(* Logix 5000 project; controller DispersionPlc vendor 1 type 14 code 108 rev 34.11; software revision 34.01; part 21 of 22 *)
(* tags used below, declared in another part *)
   DummyOutput : BOOL;
   Estop_Disp : ALIAS FOR Local:3:I.Data.1;
   FIT_4305_xx : AStd_AnalogInput;
   GenPurp : AStd_GeneralPurp;
   LS_4302_High : BOOL;
   SV_4307_1 : AStd_VlvOC;
   SV_4307_1_AOI : AStd_VlvOC_AOI;
   T0110_PhaseTimedAgitate : AStd_PLI;
   TIT_4305_1 : AStd_AnalogInput;
   TIT_4307_1 : AStd_AnalogInput;
   TIT_4307_1_AOI : AStd_AI_AOI;
   V4307_PhaseAddRO : AStd_PLI;
   V4307_PhaseAddRO_AOI : AStd_PLI_AOI;
   V4307_PhaseAgitation : AStd_PLI;
   V4307_PhaseAgitation_AOI : AStd_PLI_AOI;
   VFD_4307_1 : AStd_VFD;
   VFD_4307_1_AOI : AStd_VFD_AOI;
   WIT_4302_1 : AStd_AnalogInput;
   WIT_4307_1 : AStd_AnalogInput;
   WIT_4307_1_AOI : AStd_AI_AOI;
   XV_4301_8 : AStd_VlvOC;
   XV_4302_10 : AStd_VlvOC;
   XV_4302_8 : AStd_VlvOC;
   XV_4306_3 : AStd_VlvOC;
   XV_4306_5 : AStd_VlvOC;
   XV_4307_1 : AStd_VlvOC;
   XV_4307_1_AOI : AStd_VlvOC_AOI;
   XV_4307_1_IOpn : BOOL;
   XV_4307_1_OCls : BOOL;
   XV_4307_2 : AStd_VlvOC;
   XV_4307_2_AOI : AStd_VlvOC_AOI;
   XV_4307_2_IOpn : BOOL;
   XV_4307_2_OCls : BOOL;
   XV_4307_3 : AStd_VlvOC;
   XV_4307_3_AOI : AStd_VlvOC_AOI;
   XV_4307_3_IOpn : BOOL;
   XV_4307_3_OCls : BOOL;
   XV_4307_4 : AStd_VlvOC;
   XV_4307_4_AOI : AStd_VlvOC_AOI;
   XV_4307_4_IOpn : BOOL;
   XV_4307_4_OCls : BOOL;
   XV_4307_6 : AStd_VlvOC;
   XV_4307_6_AOI : AStd_VlvOC_AOI;
   XV_4307_6_IOpn : BOOL;
   XV_4307_6_OCls : BOOL;

PROGRAM Unit_V4307   (* main routine MainRoutine *)

ROUTINE Device_SV_4307_1   (* ladder *)
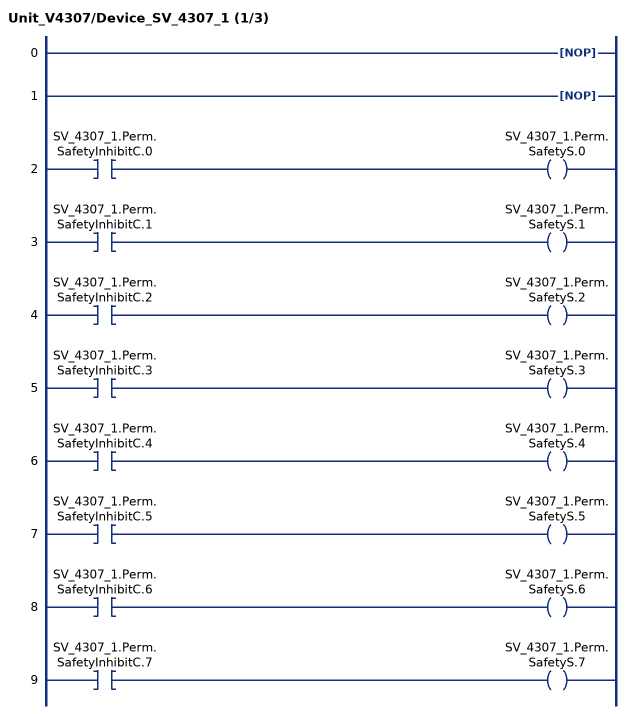
   0: NOP();
   1: NOP();
   2: XIC(SV_4307_1.Perm.SafetyInhibitC.0)OTE(SV_4307_1.Perm.SafetyS.0);
   3: XIC(SV_4307_1.Perm.SafetyInhibitC.1)OTE(SV_4307_1.Perm.SafetyS.1);
   4: XIC(SV_4307_1.Perm.SafetyInhibitC.2)OTE(SV_4307_1.Perm.SafetyS.2);
   5: XIC(SV_4307_1.Perm.SafetyInhibitC.3)OTE(SV_4307_1.Perm.SafetyS.3);
   6: XIC(SV_4307_1.Perm.SafetyInhibitC.4)OTE(SV_4307_1.Perm.SafetyS.4);
   7: XIC(SV_4307_1.Perm.SafetyInhibitC.5)OTE(SV_4307_1.Perm.SafetyS.5);
   8: XIC(SV_4307_1.Perm.SafetyInhibitC.6)OTE(SV_4307_1.Perm.SafetyS.6);
   9: XIC(SV_4307_1.Perm.SafetyInhibitC.7)OTE(SV_4307_1.Perm.SafetyS.7);
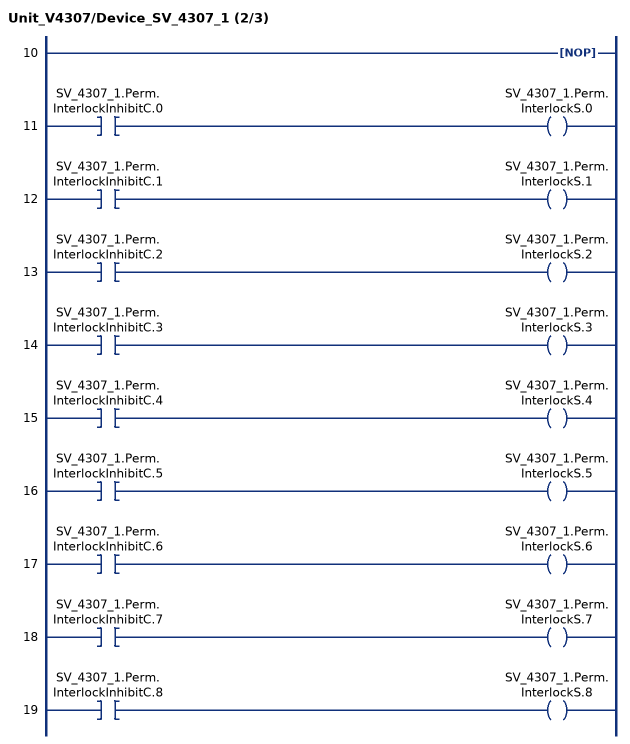
   10: NOP();
   11: XIC(SV_4307_1.Perm.InterlockInhibitC.0)OTE(SV_4307_1.Perm.InterlockS.0);
   12: XIC(SV_4307_1.Perm.InterlockInhibitC.1)OTE(SV_4307_1.Perm.InterlockS.1);
   13: XIC(SV_4307_1.Perm.InterlockInhibitC.2)OTE(SV_4307_1.Perm.InterlockS.2);
   14: XIC(SV_4307_1.Perm.InterlockInhibitC.3)OTE(SV_4307_1.Perm.InterlockS.3);
   15: XIC(SV_4307_1.Perm.InterlockInhibitC.4)OTE(SV_4307_1.Perm.InterlockS.4);
   16: XIC(SV_4307_1.Perm.InterlockInhibitC.5)OTE(SV_4307_1.Perm.InterlockS.5);
   17: XIC(SV_4307_1.Perm.InterlockInhibitC.6)OTE(SV_4307_1.Perm.InterlockS.6);
   18: XIC(SV_4307_1.Perm.InterlockInhibitC.7)OTE(SV_4307_1.Perm.InterlockS.7);
   19: XIC(SV_4307_1.Perm.InterlockInhibitC.8)OTE(SV_4307_1.Perm.InterlockS.8);
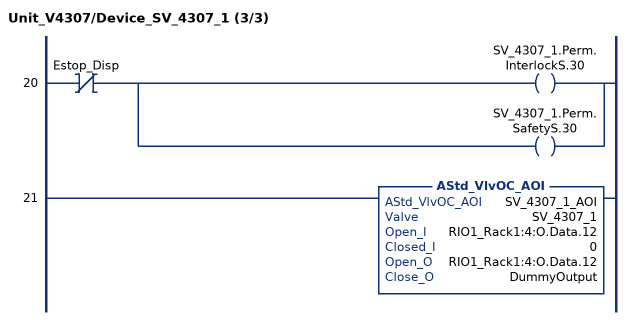
   20: XIO(Estop_Disp)[OTE(SV_4307_1.Perm.InterlockS.30) ,OTE(SV_4307_1.Perm.SafetyS.30) ];
   21: AStd_VlvOC_AOI(SV_4307_1_AOI,SV_4307_1,RIO1_Rack1:4:O.Data.12,0,RIO1_Rack1:4:O.Data.12,DummyOutput);
END_ROUTINE

ROUTINE Device_TIT_4307_1   (* ladder *)
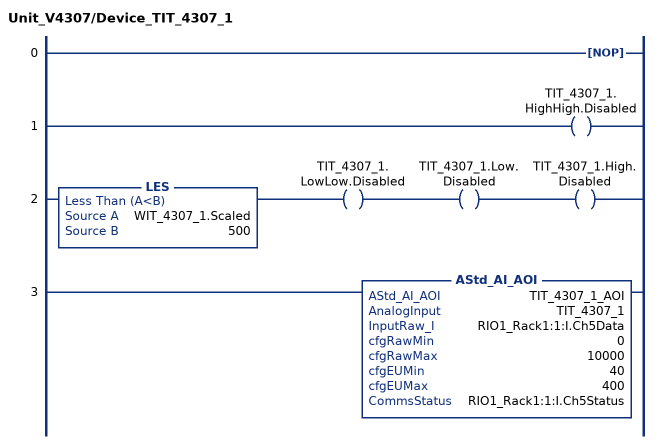
   0: NOP();
   1: OTE(TIT_4307_1.HighHigh.Disabled);
   2: LES(WIT_4307_1.Scaled,500)OTE(TIT_4307_1.LowLow.Disabled)OTE(TIT_4307_1.Low.Disabled)OTE(TIT_4307_1.High.Disabled);
   3: AStd_AI_AOI(TIT_4307_1_AOI,TIT_4307_1,RIO1_Rack1:1:I.Ch5Data,0,10000,40,400,RIO1_Rack1:1:I.Ch5Status);
END_ROUTINE

ROUTINE Device_VFD_4307_1   (* ladder *)
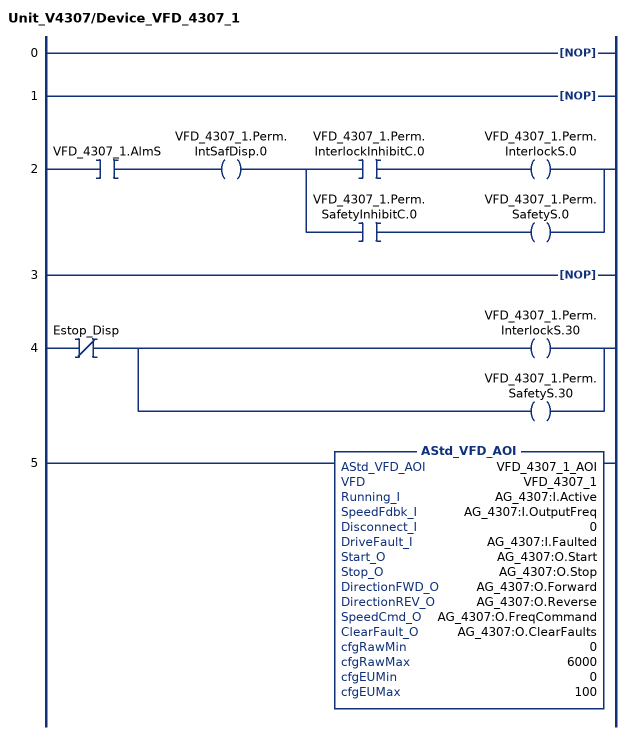
   0: NOP();
   1: NOP();
   2: XIC(VFD_4307_1.AlmS)OTE(VFD_4307_1.Perm.IntSafDisp.0)[XIC(VFD_4307_1.Perm.InterlockInhibitC.0) OTE(VFD_4307_1.Perm.InterlockS.0) ,XIC(VFD_4307_1.Perm.SafetyInhibitC.0) OTE(VFD_4307_1.Perm.SafetyS.0) ];
   3: NOP();
   4: XIO(Estop_Disp)[OTE(VFD_4307_1.Perm.InterlockS.30) ,OTE(VFD_4307_1.Perm.SafetyS.30) ];
   5: AStd_VFD_AOI(VFD_4307_1_AOI,VFD_4307_1,AG_4307:I.Active,AG_4307:I.OutputFreq,0,AG_4307:I.Faulted,AG_4307:O.Start,AG_4307:O.Stop,AG_4307:O.Forward,AG_4307:O.Reverse,AG_4307:O.FreqCommand,AG_4307:O.ClearFaults,0,6000,0,100);
END_ROUTINE

ROUTINE Device_WIT_4307_1   (* ladder *)
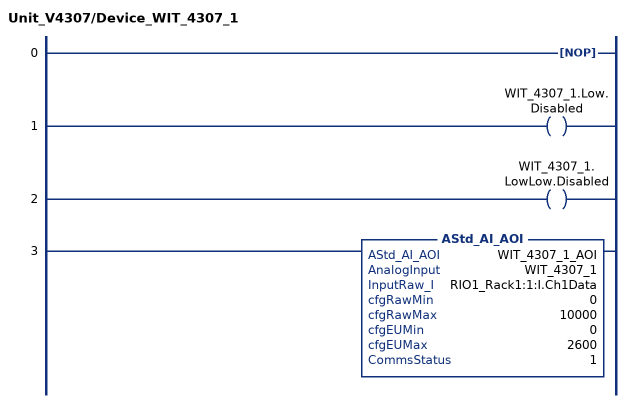
   0: NOP();
   1: OTE(WIT_4307_1.Low.Disabled);
   2: OTE(WIT_4307_1.LowLow.Disabled);
   3: AStd_AI_AOI(WIT_4307_1_AOI,WIT_4307_1,RIO1_Rack1:1:I.Ch1Data,0,10000,0,2600,1);
END_ROUTINE

ROUTINE Device_XV_4307_1   (* ladder *)
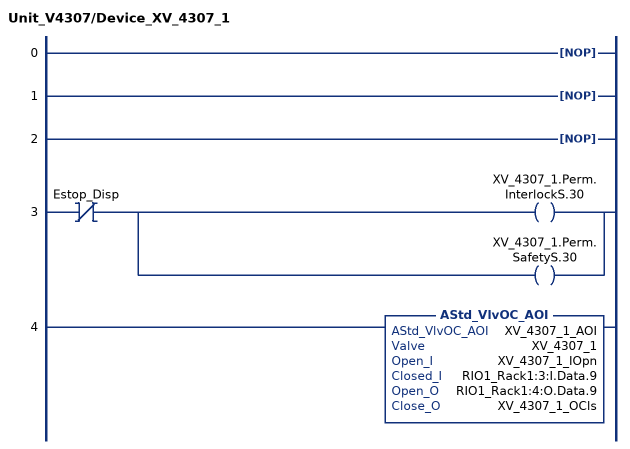
   0: NOP();
   1: NOP();
   2: NOP();
   3: XIO(Estop_Disp)[OTE(XV_4307_1.Perm.InterlockS.30) ,OTE(XV_4307_1.Perm.SafetyS.30) ];
   4: AStd_VlvOC_AOI(XV_4307_1_AOI,XV_4307_1,XV_4307_1_IOpn,RIO1_Rack1:3:I.Data.9,RIO1_Rack1:4:O.Data.9,XV_4307_1_OCls);
END_ROUTINE

ROUTINE Device_XV_4307_2   (* ladder *)
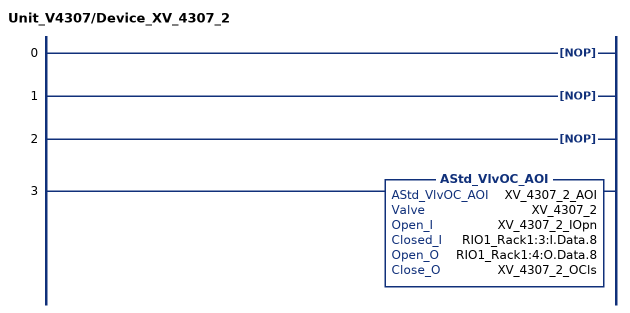
   0: NOP();
   1: NOP();
   2: NOP();
   3: AStd_VlvOC_AOI(XV_4307_2_AOI,XV_4307_2,XV_4307_2_IOpn,RIO1_Rack1:3:I.Data.8,RIO1_Rack1:4:O.Data.8,XV_4307_2_OCls);
END_ROUTINE

ROUTINE Device_XV_4307_3   (* ladder *)
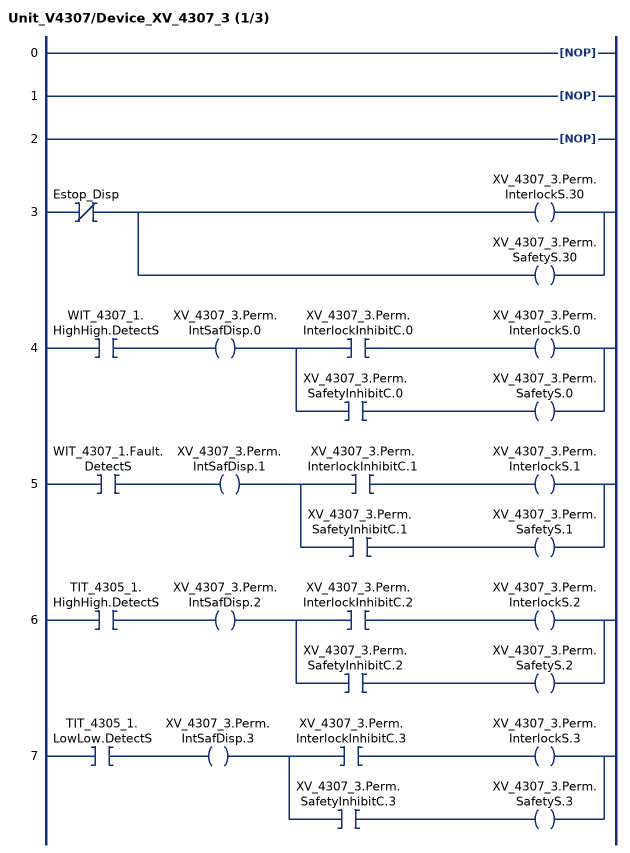
   0: NOP();
   1: NOP();
   2: NOP();
   3: XIO(Estop_Disp)[OTE(XV_4307_3.Perm.InterlockS.30) ,OTE(XV_4307_3.Perm.SafetyS.30) ];
   4: XIC(WIT_4307_1.HighHigh.DetectS)OTE(XV_4307_3.Perm.IntSafDisp.0)[XIC(XV_4307_3.Perm.InterlockInhibitC.0) OTE(XV_4307_3.Perm.InterlockS.0) ,XIC(XV_4307_3.Perm.SafetyInhibitC.0) OTE(XV_4307_3.Perm.SafetyS.0) ];
   5: XIC(WIT_4307_1.Fault.DetectS)OTE(XV_4307_3.Perm.IntSafDisp.1)[XIC(XV_4307_3.Perm.InterlockInhibitC.1) OTE(XV_4307_3.Perm.InterlockS.1) ,XIC(XV_4307_3.Perm.SafetyInhibitC.1) OTE(XV_4307_3.Perm.SafetyS.1) ];
   6: XIC(TIT_4305_1.HighHigh.DetectS)OTE(XV_4307_3.Perm.IntSafDisp.2)[XIC(XV_4307_3.Perm.InterlockInhibitC.2) OTE(XV_4307_3.Perm.InterlockS.2) ,XIC(XV_4307_3.Perm.SafetyInhibitC.2) OTE(XV_4307_3.Perm.SafetyS.2) ];
   7: XIC(TIT_4305_1.LowLow.DetectS)OTE(XV_4307_3.Perm.IntSafDisp.3)[XIC(XV_4307_3.Perm.InterlockInhibitC.3) OTE(XV_4307_3.Perm.InterlockS.3) ,XIC(XV_4307_3.Perm.SafetyInhibitC.3) OTE(XV_4307_3.Perm.SafetyS.3) ];
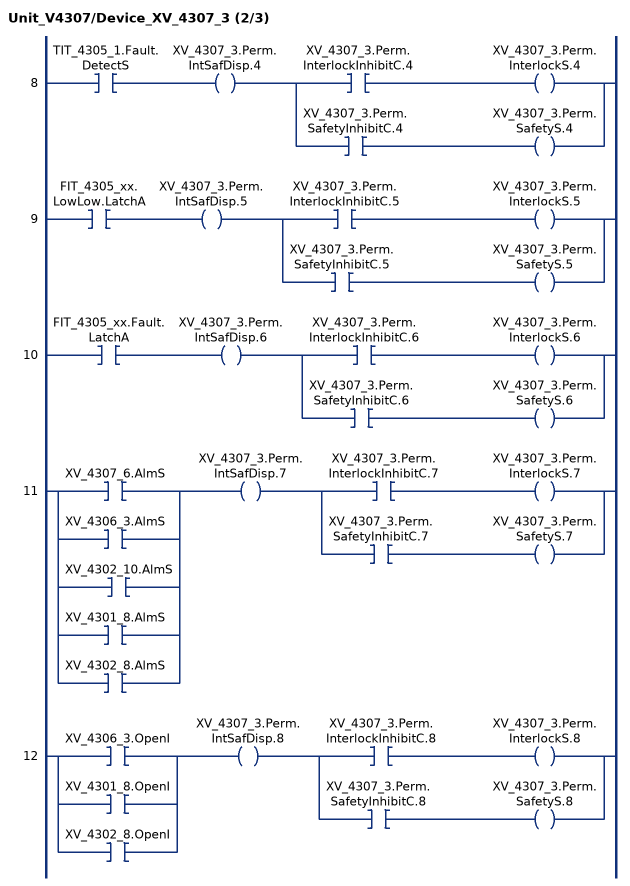
   8: XIC(TIT_4305_1.Fault.DetectS)OTE(XV_4307_3.Perm.IntSafDisp.4)[XIC(XV_4307_3.Perm.InterlockInhibitC.4) OTE(XV_4307_3.Perm.InterlockS.4) ,XIC(XV_4307_3.Perm.SafetyInhibitC.4) OTE(XV_4307_3.Perm.SafetyS.4) ];
   9: XIC(FIT_4305_xx.LowLow.LatchA)OTE(XV_4307_3.Perm.IntSafDisp.5)[XIC(XV_4307_3.Perm.InterlockInhibitC.5) OTE(XV_4307_3.Perm.InterlockS.5) ,XIC(XV_4307_3.Perm.SafetyInhibitC.5) OTE(XV_4307_3.Perm.SafetyS.5) ];
   10: XIC(FIT_4305_xx.Fault.LatchA)OTE(XV_4307_3.Perm.IntSafDisp.6)[XIC(XV_4307_3.Perm.InterlockInhibitC.6) OTE(XV_4307_3.Perm.InterlockS.6) ,XIC(XV_4307_3.Perm.SafetyInhibitC.6) OTE(XV_4307_3.Perm.SafetyS.6) ];
   11: [XIC(XV_4307_6.AlmS) ,XIC(XV_4306_3.AlmS) ,XIC(XV_4302_10.AlmS) ,XIC(XV_4301_8.AlmS) ,XIC(XV_4302_8.AlmS) ]OTE(XV_4307_3.Perm.IntSafDisp.7)[XIC(XV_4307_3.Perm.InterlockInhibitC.7) OTE(XV_4307_3.Perm.InterlockS.7) ,XIC(XV_4307_3.Perm.SafetyInhibitC.7) OTE(XV_4307_3.Perm.SafetyS.7) ];
   12: [XIC(XV_4306_3.OpenI) ,XIC(XV_4301_8.OpenI) ,XIC(XV_4302_8.OpenI) ]OTE(XV_4307_3.Perm.IntSafDisp.8)[XIC(XV_4307_3.Perm.InterlockInhibitC.8) OTE(XV_4307_3.Perm.InterlockS.8) ,XIC(XV_4307_3.Perm.SafetyInhibitC.8) OTE(XV_4307_3.Perm.SafetyS.8) ];
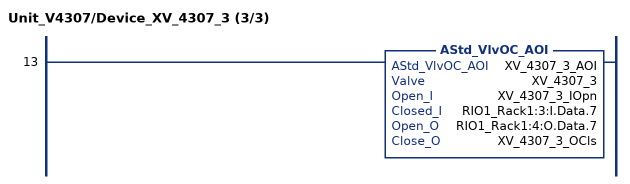
   13: AStd_VlvOC_AOI(XV_4307_3_AOI,XV_4307_3,XV_4307_3_IOpn,RIO1_Rack1:3:I.Data.7,RIO1_Rack1:4:O.Data.7,XV_4307_3_OCls);
END_ROUTINE

ROUTINE Device_XV_4307_4   (* ladder *)
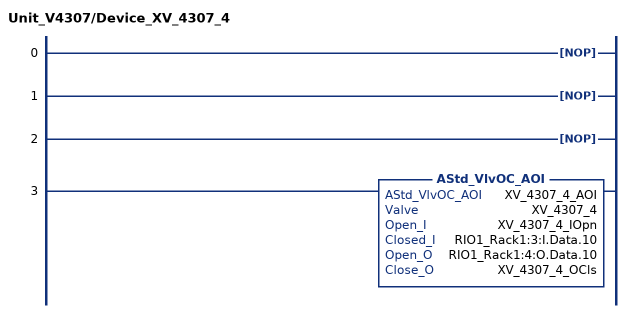
   0: NOP();
   1: NOP();
   2: NOP();
   3: AStd_VlvOC_AOI(XV_4307_4_AOI,XV_4307_4,XV_4307_4_IOpn,RIO1_Rack1:3:I.Data.10,RIO1_Rack1:4:O.Data.10,XV_4307_4_OCls);
END_ROUTINE

ROUTINE Device_XV_4307_6   (* ladder *)
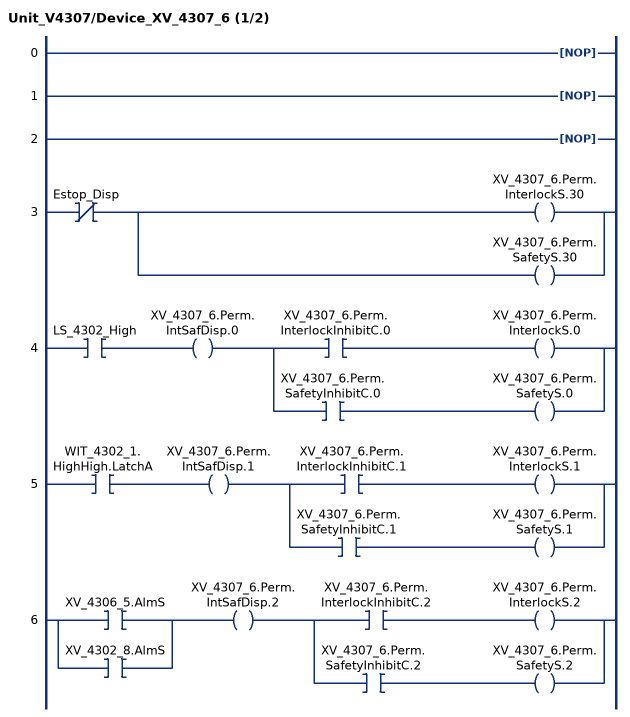
   0: NOP();
   1: NOP();
   2: NOP();
   3: XIO(Estop_Disp)[OTE(XV_4307_6.Perm.InterlockS.30) ,OTE(XV_4307_6.Perm.SafetyS.30) ];
   4: XIC(LS_4302_High)OTE(XV_4307_6.Perm.IntSafDisp.0)[XIC(XV_4307_6.Perm.InterlockInhibitC.0) OTE(XV_4307_6.Perm.InterlockS.0) ,XIC(XV_4307_6.Perm.SafetyInhibitC.0) OTE(XV_4307_6.Perm.SafetyS.0) ];
   5: XIC(WIT_4302_1.HighHigh.LatchA)OTE(XV_4307_6.Perm.IntSafDisp.1)[XIC(XV_4307_6.Perm.InterlockInhibitC.1) OTE(XV_4307_6.Perm.InterlockS.1) ,XIC(XV_4307_6.Perm.SafetyInhibitC.1) OTE(XV_4307_6.Perm.SafetyS.1) ];
   6: [XIC(XV_4306_5.AlmS) ,XIC(XV_4302_8.AlmS) ]OTE(XV_4307_6.Perm.IntSafDisp.2)[XIC(XV_4307_6.Perm.InterlockInhibitC.2) OTE(XV_4307_6.Perm.InterlockS.2) ,XIC(XV_4307_6.Perm.SafetyInhibitC.2) OTE(XV_4307_6.Perm.SafetyS.2) ];
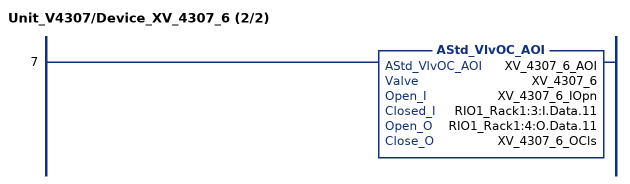
   7: AStd_VlvOC_AOI(XV_4307_6_AOI,XV_4307_6,XV_4307_6_IOpn,RIO1_Rack1:3:I.Data.11,RIO1_Rack1:4:O.Data.11,XV_4307_6_OCls);
END_ROUTINE

ROUTINE MainRoutine   (* ladder *)
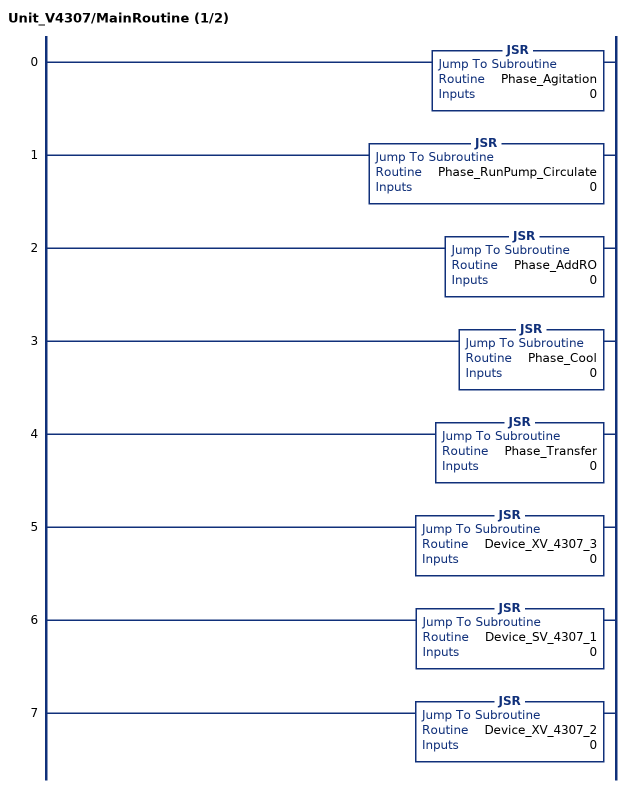
   0: JSR(Phase_Agitation,0);
   1: JSR(Phase_RunPump_Circulate,0);
   2: JSR(Phase_AddRO,0);
   3: JSR(Phase_Cool,0);
   4: JSR(Phase_Transfer,0);
   5: JSR(Device_XV_4307_3,0);
   6: JSR(Device_SV_4307_1,0);
   7: JSR(Device_XV_4307_2,0);
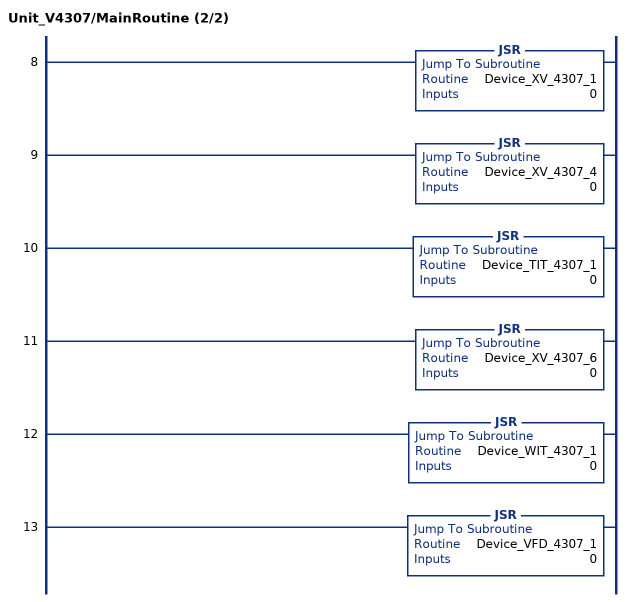
   8: JSR(Device_XV_4307_1,0);
   9: JSR(Device_XV_4307_4,0);
   10: JSR(Device_TIT_4307_1,0);
   11: JSR(Device_XV_4307_6,0);
   12: JSR(Device_WIT_4307_1,0);
   13: JSR(Device_VFD_4307_1,0);
END_ROUTINE

ROUTINE Phase_AddRO   (* ladder *)
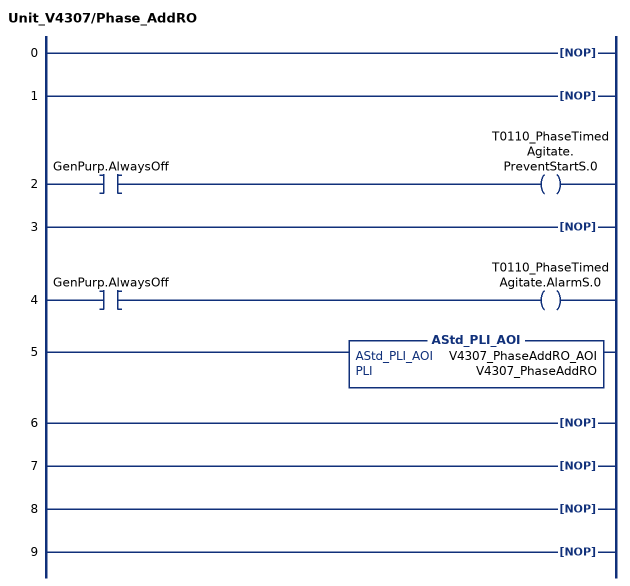
   0: NOP();
   1: NOP();
   2: XIC(GenPurp.AlwaysOff)OTE(T0110_PhaseTimedAgitate.PreventStartS.0);
   3: NOP();
   4: XIC(GenPurp.AlwaysOff)OTE(T0110_PhaseTimedAgitate.AlarmS.0);
   5: AStd_PLI_AOI(V4307_PhaseAddRO_AOI,V4307_PhaseAddRO);
   6: NOP();
   7: NOP();
   8: NOP();
   9: NOP();
END_ROUTINE

ROUTINE Phase_Agitation   (* ladder *)
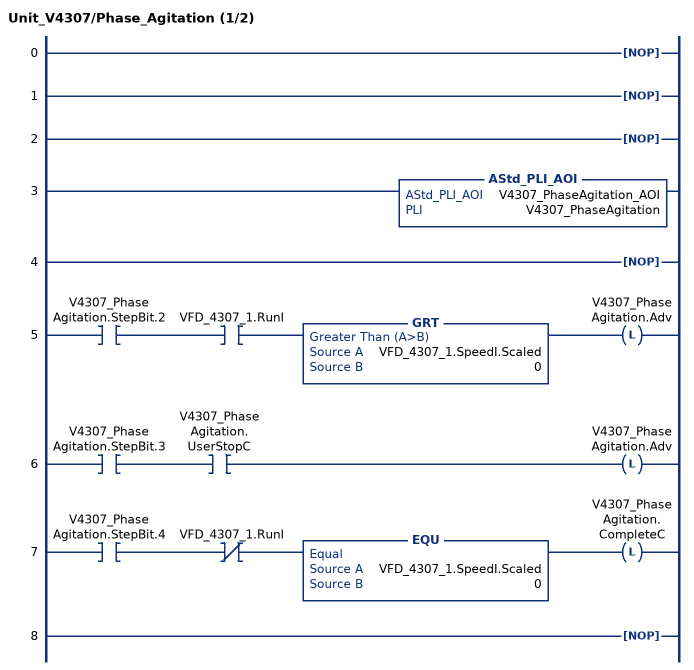
   0: NOP();
   1: NOP();
   2: NOP();
   3: AStd_PLI_AOI(V4307_PhaseAgitation_AOI,V4307_PhaseAgitation);
   4: NOP();
   5: XIC(V4307_PhaseAgitation.StepBit.2)XIC(VFD_4307_1.RunI)GRT(VFD_4307_1.SpeedI.Scaled,0)OTL(V4307_PhaseAgitation.Adv);
   6: XIC(V4307_PhaseAgitation.StepBit.3)XIC(V4307_PhaseAgitation.UserStopC)OTL(V4307_PhaseAgitation.Adv);
   7: XIC(V4307_PhaseAgitation.StepBit.4)XIO(VFD_4307_1.RunI)EQU(VFD_4307_1.SpeedI.Scaled,0)OTL(V4307_PhaseAgitation.CompleteC);
   8: NOP();
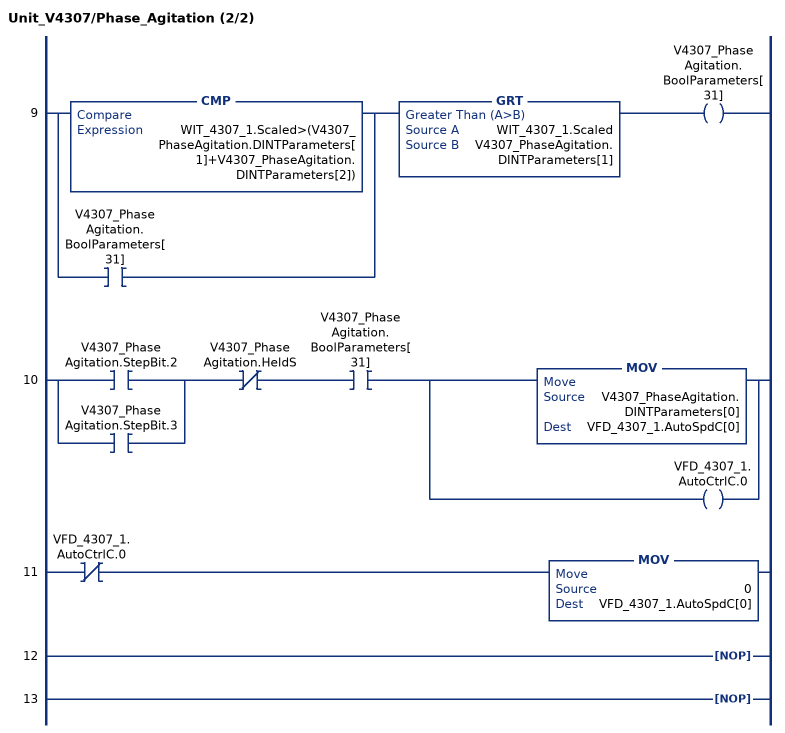
   9: [CMP(WIT_4307_1.Scaled>(V4307_PhaseAgitation.DINTParameters[1]+V4307_PhaseAgitation.DINTParameters[2])) ,XIC(V4307_PhaseAgitation.BoolParameters[31]) ]GRT(WIT_4307_1.Scaled,V4307_PhaseAgitation.DINTParameters[1])OTE(V4307_PhaseAgitation.BoolParameters[31]);
   10: [XIC(V4307_PhaseAgitation.StepBit.2) ,XIC(V4307_PhaseAgitation.StepBit.3) ]XIO(V4307_PhaseAgitation.HeldS)XIC(V4307_PhaseAgitation.BoolParameters[31])[MOV(V4307_PhaseAgitation.DINTParameters[0],VFD_4307_1.AutoSpdC[0]) ,OTE(VFD_4307_1.AutoCtrlC.0) ];
   11: XIO(VFD_4307_1.AutoCtrlC.0)MOV(0,VFD_4307_1.AutoSpdC[0]);
   12: NOP();
   13: NOP();
END_ROUTINE
